// TIA Portal V19 export
FUNCTION "Fix_Screen" : Void   // FC38, STL
{ S7_Optimized_Access := 'TRUE' }
AUTHOR : OPA_8160
FAMILY : APP
NAME : FixScre
// stored: AutoNumber false
BEGIN

NETWORK
TITLE = 
// Control variable for multiplexing variables in fixed screen on OP25
// Fixed Screen on OP25 is toggling between TANK and UHT-PLC
      L     "Tag_75";
      L     10;  // SCREEN NUMBERS < 10 BELONGS TO SYSTEM SCREENS
      <=I;  // IF A SYSTEM SCREEN IS SELECTED
      BEC;  // KEEP FIXED SCEEN FROM PREVIOUS STATE
      L     "Tag_75";
      L     50;
      >I;
      JC    C001;
      S     "ViewUHT_TANK_OP25";  // VIEW FILLER STATUS IN FIXED SCREEN
      L     1;
      T     "Tag_76";
      BEC;
C001: NOP   0;
      R     "ViewUHT_TANK_OP25";  // VIEW ASEPTIC TANK STATUS IN FIXED SCREEN
      L     0;
      T     "Tag_76";
END_FUNCTION
